{attribute 'qualified_only'}
VAR_GLOBAL
	{attribute 'OPC.UA.DA.StructuredType' := '1'}
	{attribute 'OPC.UA.DA' := '1'}
	ROB : ARRAY[1..3] of FB_ROB;
END_VAR

(* stored: Version 1.1.0.1, ProductVersion 3.1.4026.18
   GVL OPCUA: Id {817fe7bd-fd4a-490a-a2c0-af3e328eba30} *)
